// Digital output group
FUNCTION_BLOCK FB_DOGroup EXTENDS FB_IOGroup IMPLEMENTS I_DOGroup
VAR
	aOut			: ARRAY [0..nMaxSize - 1] OF I_DigitalOut;		// Array of interfaces to digital outputs
	
	aIndicator		: ARRAY [0..nMaxSize - 1] OF I_DigitalOut;		// Array of interfaces to digital outputs that serve as indicators
	nSizeIndicators	: INT;											// Size of indicator array
END_VAR

// Add indicator to group.
// Indicators are defined separately from outputs. Indicators follow outputs and the link between them is defined in the PLC.
// Regardless of how the output is updated (by the PLC or externally), the indicators follow the outputs. 
METHOD AddIndicator
VAR_INPUT
	IDO			: I_DigitalOut;		// Interface to digital output that needs to be an indicator
END_VAR
IF nSizeIndicators < nMaxSize THEN
	aIndicator[nSizeIndicators] := IDO;
	nSizeIndicators := nSizeIndicators + 1;
END_IF
END_METHOD

// Add output to group
METHOD AddOutput
VAR_INPUT
	IDO			: I_DigitalOut;		// Interface to digital output
END_VAR
IF nSize < nMaxSize THEN
	aOut[nSize] := IDO;
	nSize := nSize + 1;
END_IF
END_METHOD

// Runs the execute method of all digital output FBs in the group.
// Make sure all digital output execute methods are called only once per PLC cyle
METHOD Execute
VAR
	i		: INT;		// Iterator variable
END_VAR
// Call the execute method of all digital outputs in the group
FOR i := 0 TO nSize - 1 DO
	aOut[i].Execute();
END_FOR
END_METHOD

// Get a specific output from the group
METHOD GetOutput : I_DigitalOut
VAR_INPUT
	nOutputIndex		: INT;		// Output index
END_VAR
GetOutput := aOut[nOutputIndex];
END_METHOD

// Set the command to the outputs in the group
METHOD SetCommand
VAR_INPUT
	eCommand	: E_DOCommand;
END_VAR
VAR
	i			: INT;
END_VAR
FOR i := 0 TO nSize - 1 DO
	IF aOut[i].Command = E_DOCommand.None THEN
		// No command yet, set new command
		aOut[i].SetCommand(eCommand);
	ELSE
		// A command was already issued
		// Do nothing
	END_IF
END_FOR
END_METHOD

// Update the indicator values based on the value of the outputs
METHOD UpdateIndicators
VAR
	i	: INT;		// Iterator variable
END_VAR
// Check if there is at least one output in the group since at least one output is needed to determine the output value
IF nSize > 0 THEN
	// Set output value of all indicators to that of the first output in the group (all others are the same anyway)
	FOR i := 0 TO nSizeIndicators - 1 DO
		aIndicator[i].Output := aOut[0].Output;
	END_FOR
END_IF
END_METHOD

END_FUNCTION_BLOCK

(* stored: Version 1.1.0.1, ProductVersion 3.1.4024.12
   POU FB_DOGroup: Id {b3488830-ec61-443c-9742-10099d09d800}, SpecialFunc None
   Folder Methods: Id {3a95f167-8838-43a7-9c46-3573e393aca1}
   Method AddIndicator: Id {0d2a6617-311a-4efc-96e6-1ebf7609d9f7}
   Method AddOutput: Id {d02ea73d-8c89-4a2a-8090-763a0721398e}
   Method Execute: Id {e77e7b2c-f6f1-456d-bfbf-b27bf30a79b9}
   Method GetOutput: Id {3ab7d26e-6f1d-4872-b024-6588ee0cb538}
   Method SetCommand: Id {9ed0280c-8f0a-4e75-8f4b-35a22c587e1b}
   Method UpdateIndicators: Id {c2af6b2e-8e0c-4bed-815d-f454ed6e90fb} *)
